PROGRAM Func_example
VAR
	iMyInt : INT;
	uMyInt : INT;
	TmpC : LREAL;
	TmpF : LREAL;
END_VAR

iMyInt := UINT_TO_INT(uMyInt);

TmpF := F_CtoF(TmpC);

END_PROGRAM

(* stored: Version 1.1.0.1, ProductVersion 3.1.4024.9
   POU Func_example: Id {20b0ab15-9e17-449f-8193-f66a1969e117}, SpecialFunc None *)
